// TIA Portal V15.1 export
// export: Created 2026-01-15T16:29:41.8073062Z, ExportSetting WithDefaults, WithReadOnly, DisplayName Totally Integrated Automation Portal, DisplayVersion V15.1 Update 8, DisplayName TIA Portal Openness, DisplayVersion V15.1 Update 8, DisplayName STEP 7 Professional, DisplayVersion V15.1 Update 8, DisplayName WinCC Advanced, DisplayVersion V15.1 Update 8
DATA_BLOCK "4.SIMULATION"   // DB400
{ S7_Optimized_Access := 'TRUE' }
VERSION : 0.1
// stored: AutoNumber false, CodeModifiedDate 2026-01-15T16:25:55.15091Z, CompileDate 2026-01-15T16:25:55.1580097Z, CreationDate 2026-01-15T16:22:49.8270549Z, DBAccessibleFromOPCUA true, DownloadWithoutReinit false, InstanceOfName 4.SIMULATION_DATA, InstanceOfNumber 4, InstanceOfType FB, InterfaceModifiedDate 2023-11-28T22:28:44.2264332Z, IsConsistent true, IsKnowHowProtected false, IsRetainMemResEnabled false, MemoryReserve 100, ModifiedDate 2026-01-15T16:25:55.15091Z, ParameterModified 2023-11-28T22:28:44.2264332Z, StructureModified 2023-11-28T22:28:44.2264332Z, UDAEnableTagReadback false
"4.SIMULATION_DATA"
   // VAR_INPUT
   //    RE_SET : Bool;
   //    XUNG_CLOCK : Bool;
   //    CAN_1 : Bool;
   //    CAN_2 : Bool;
   //    CAN_3 : Bool;
   //    CAN_4 : Bool;
   //    CAN_5 : Bool;
   //    CAN_6 : Bool;
   //    CAN_7 : Bool;
   //    CAN_8 : Bool;
   //    CAN_9 : Bool;
   //    CAN_10 : Bool;
   //    CAN_11 : Bool;
   //    CAN_12 : Bool;
   //    XA_1 : Bool;
   //    XA_2 : Bool;
   //    XA_3 : Bool;
   //    XA_4 : Bool;
   //    XA_5 : Bool;
   //    XA_6 : Bool;
   //    XA_7 : Bool;
   //    XA_8 : Bool;
   //    XA_9 : Bool;
   //    XA_10 : Bool;
   //    XA_11 : Bool;
   //    XA_12 : Bool;
   //    HS_NAP_AGG1 : Real;
   //    HS_NAP_AGG2 : Real;
   //    HS_NAP_AGG3 : Real;
   //    HS_NAP_AGG4 : Real;
   //    HS_NAP_AGG5 : Real;
   //    HS_NAP_AGG6 : Real;
   //    HS_NAP_CEM1 : Real;
   //    HS_NAP_CEM2 : Real;
   //    HS_NAP_WAT1 : Real;
   //    HS_NAP_WAT2 : Real;
   //    HS_NAP_ADD1 : Real;
   //    HS_NAP_ADD2 : Real;
   //    HS_XA_AGG1 : Real;
   //    HS_XA_AGG2 : Real;
   //    HS_XA_AGG3 : Real;
   //    HS_XA_AGG4 : Real;
   //    HS_XA_AGG5 : Real;
   //    HS_XA_AGG6 : Real;
   //    HS_XA_CEM1 : Real;
   //    HS_XA_CEM2 : Real;
   //    HS_XA_WAT1 : Real;
   //    HS_XA_WAT2 : Real;
   //    HS_XA_ADD1 : Real;
   //    HS_XA_ADD2 : Real;
   // END_VAR
   // VAR_OUTPUT
   //    AGG1 : Real;
   //    AGG2 : Real;
   //    AGG3 : Real;
   //    AGG4 : Real;
   //    AGG5 : Real;
   //    AGG6 : Real;
   //    CEM1 : Real;
   //    CEM2 : Real;
   //    WAT1 : Real;
   //    WAT2 : Real;
   //    WADD1 : Real;
   //    WADD2 : Real;
   // END_VAR
   // VAR
   //    A1 : Bool;
   //    B1 : Bool;
   //    A2 : Bool;
   //    B2 : Bool;
   //    A3 : Bool;
   //    B3 : Bool;
   //    A4 : Bool;
   //    B4 : Bool;
   //    A5 : Bool;
   //    B5 : Bool;
   //    A6 : Bool;
   //    B6 : Bool;
   //    A7 : Bool;
   //    B7 : Bool;
   //    A8 : Bool;
   //    B8 : Bool;
   //    A9 : Bool;
   //    B9 : Bool;
   //    A10 : Bool;
   //    B10 : Bool;
   //    A11 : Bool;
   //    B11 : Bool;
   //    A12 : Bool;
   //    B12 : Bool;
   // END_VAR
BEGIN
END_DATA_BLOCK
